Fanuc KAREL source: kc00013.KL

PROGRAM KC00013
%STACKSIZE=65535
%PRIORITY=65535
%NOLOCKGROUP
VAR
I : INTEGER
J : INTEGER
K : INTEGER
R : REAL
B : BOOLEAN
S : STRING[80]
T : STRING[80]
AI : ARRAY[8] OF INTEGER
-- UNRESOLVED DECLARATIONS (source type spelling not recovered)
-- P : TYPE_0x001F (type_u16=0x001F)
-- Q : TYPE_0x001F (type_u16=0x001F)
-- QT : TYPE_0x1102 (type_u16=0x1102)
-- AB : ARRAY[244] OF TYPE_0x0018 (type_u16=0x2018)
BEGIN
GET_QUEUE(QT,AI,I,J,K)
END KC00013
